PROGRAM Group_Template
VAR
	//iSetGroupNumber : INT := 1; //SET THIS TO THE NUMBER FOR THIS GROUP
END_VAR

//Sample code for defining groups by iterating through each axis on startup and adding all matching axis to this array
(*
IF _TaskInfo[fbGetCurTaskIndex.index].FirstCycle THEN
	GVL.iAxesGroupIndex := 1;
	FOR GVL.iAxis := 1 TO GVL_APP.nAXIS_NUM DO
		IF astAxesLocal[GVL.iAxis].stDescription.iGroupNumber = iSetGroupNumber THEN
			GVL.astAxesLocalGroup[iSetGroupNumber].aAxesInGroup[GVL.iAxesGroupIndex] := UINT_TO_INT(GVL.iAxis);
			GVL.iAxesGroupIndex := GVL.iAxesGroupIndex + 1;
		END_IF
	END_FOR
	GVL.astAxesLocalGroup[iSetGroupNumber].stDescription.iAxesInGroup := GVL.iAxesGroupIndex -1;
END_IF
*)

END_PROGRAM

(* stored: Version 1.1.0.1, ProductVersion 3.1.4026.18
   POU Group_Template: Id {d96a96f7-3990-4cce-8452-f53b9c3154ba}, SpecialFunc None *)
